// TwinCAT 3 PLC project Main
// ProgramVersion: 3.1.4023.0
// libraries:
//   Tc2_Standard, * (Beckhoff Automation GmbH)
//   Tc2_System, * (Beckhoff Automation GmbH)
//   Tc3_Module, * (Beckhoff Automation GmbH)
//   TcUnit, * (www.tcunit.org)
//   mobject-disposable,1.1.1,mobject
// project tree:
//   / PlcTask.TcTTO
//   POUs/ MAIN.TcPOU
//   Tests/ Disposable_TestSuite.TcPOU
//   Tests/Mocks/ MockDisposable.TcPOU
// real-time tasks:
//   TASK PlcTask: cycle T#10ms, priority 20, ADS port 350

CONFIGURATION Main
    RESOURCE PLC ON TwinCAT3
        TASK PlcTask(INTERVAL := T#10ms, PRIORITY := 20);
        PROGRAM MAIN WITH PlcTask : MAIN;
    END_RESOURCE
END_CONFIGURATION

// ---- POUs/MAIN.TcPOU
PROGRAM MAIN
VAR
	disposable_TestSuite : Disposable_TestSuite;
END_VAR

TcUnit.RUN();

END_PROGRAM

// ---- Tests/Disposable_TestSuite.TcPOU
FUNCTION_BLOCK PUBLIC Disposable_TestSuite EXTENDS TcUnit.FB_TestSuite
VAR
END_VAR

DisposedFromDisposeMethod();
DisposedByManuallyDeleting();

METHOD PUBLIC DisposedByManuallyDeleting
VAR
	mockDispose : POINTER TO MockDisposable;
	disposed : BOOL;
END_VAR
TEST('DisposedByManuallyDeleting');

// @TEST-FIXTURE
mockDispose := __NEW(MockDisposable(DisposedFlag:=disposed));

// @TEST-RUN
__DELETE(mockDispose);

// @TEST-ASSSERT
AssertTrue(
	Condition := disposed,
	Message := 'FB_exit was not correctly triggered in the MockDisposable'
);

TEST_FINISHED();
END_METHOD

METHOD PUBLIC DisposedFromDisposeMethod
VAR
	mockDispose : POINTER TO MockDisposable;
	disposed : BOOL;
END_VAR
TEST('DisposedFromDisposeMethod');

// @TEST-FIXTURE
mockDispose := __NEW(MockDisposable(DisposedFlag:=disposed));

// @TEST-RUN
mockDispose^.Dispose();

// @TEST-ASSSERT
AssertTrue(
	Condition := disposed,
	Message := 'FB_exit was not correctly triggered in the MockDisposable'
);

TEST_FINISHED();
END_METHOD

END_FUNCTION_BLOCK

// ---- Tests/Mocks/MockDisposable.TcPOU
{attribute 'linkalways'} 
{attribute 'no_explicit_call' := 'This FB is a CLASS and must be accessed using methods or properties'}
{attribute 'enable_dynamic_creation'}
FUNCTION_BLOCK MockDisposable EXTENDS Disposable
VAR
	disposedFlag : REFERENCE TO BOOL;
END_VAR

METHOD FB_exit : BOOL
VAR_INPUT
	bInCopyCode : BOOL; // if TRUE, the exit method is called for exiting an instance that is copied afterwards (online change).
END_VAR
disposedFlag := TRUE;
END_METHOD

METHOD FB_init : BOOL
VAR_INPUT
	bInitRetains : BOOL; // if TRUE, the retain variables are initialized (warm start / cold start)
	bInCopyCode : BOOL;  // if TRUE, the instance afterwards gets moved into the copy code (online change)
	DisposedFlag : REFERENCE TO BOOL;
END_VAR
THIS^.disposedFlag REF= DisposedFlag;
END_METHOD

END_FUNCTION_BLOCK
